// Mitsubishi GX Works2 project: 이중 코일   PLC: Q03UDV

PROGRAM MAIN
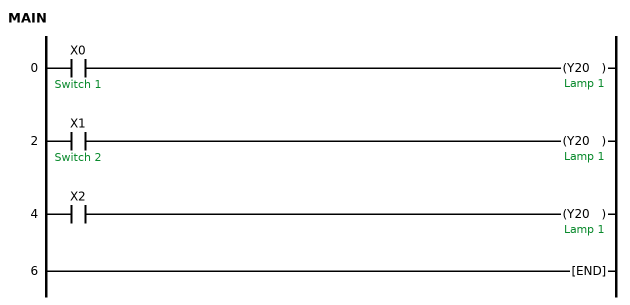
0     LD      X0  ; Switch 1
      OUT     Y20  ; Lamp 1
2     LD      X1  ; Switch 2
      OUT     Y20  ; Lamp 1
4     LD      X2
      OUT     Y20  ; Lamp 1
6     END
END_PROGRAM
